TYPE E_ExchangePieceOption :
(
	Slot := 0,
	NextSlotRespPiece := 1
)USINT;
END_TYPE

(* stored: Version 1.1.0.1, ProductVersion 3.1.0.25
   DUT E_ExchangePieceOption: Id {bf5ae7d3-9a94-4139-940b-5755eba209d0} *)
